# EPICS substitutions: hugo/source/db/Beckhoff_6XXX/ecmcEL6080.substitutions
file "ecmcEL6080-chX.template"
{
  pattern {}
          {}
}
